(* LS Electric XG5000 project: XEM_iX7_ModTCP_Example *)
(* PLC LSPLC *)
(* module base 0 slot 0: Input/Output Module:XEM-DN/DP32HP (DC 24V Input, Transistor Output, 32 Contacts) *)
(* module base 0 slot 1: Internal Positioning:XBF-PO06E (Open Collector Type, 6 Axis) *)
VAR_GLOBAL
    gControl_Word AT %MW1 : WORD; (* global control word for controlling the iX7 over Modbus TCP *)
    gStatus_Word AT %MW2 : WORD; (* global status word data for iX7 drive over Modbus TCP *)
    gSV_ON AT %MX0 : BOOL; (* global Command to turn servo on/off sent over Modbus RTU *)
    gTarget_Position AT %MW3 : ARRAY[0..1] OF WORD; (* global target position in an array of words *)
    gVelocity_Accel_Decel AT %MW4 : ARRAY[0..5] OF WORD; (* word array for setting up velocity, acceleration and deceleration of the modbus TCP move *)
END_VAR

PROGRAM NewProgram (* task: Scan Program *)
VAR
    Acceleration : DINT; (* acceleration of the move *)
    Deceleration : DINT; (* deceleration of the move *)
    Halt_Motion : BOOL; (* halt motion of the modbus servo *)
    Move_Type0 : BOOL; (* Move type 0 is wait until current move is complete *)
    Move_Type1 : BOOL; (* move to target position immediately *)
    Move_Type2 : BOOL; (* Drives from the current position to the profile position at the profile / velocity before it applies the next position. *)
    Positioning_Mode : BOOL; (* False = Absolute Positioning; True = Relative Positioning *)
    Servo_Enable : BOOL; (* Enable servo - local command to enable servos *)
    Start_Motion : BOOL; (* local command to start motion *)
    Target_Position : DINT; (* local index01 distance value *)
    tempDword : DWORD; (* temporary dword storage *)
    Velocity : DINT; (* velocity of the move *)
END_VAR
VAR_EXTERNAL
    gControl_Word : WORD; (* AT %MW1 *) (* global control word for controlling the iX7 over Modbus TCP *)
    gStatus_Word : WORD; (* AT %MW2 *) (* global status word data for iX7 drive over Modbus TCP *)
    gSV_ON : BOOL; (* AT %MX0 *) (* global Command to turn servo on/off sent over Modbus RTU *)
    gTarget_Position : ARRAY[0..1] OF WORD; (* AT %MW3 *) (* global target position in an array of words *)
    gVelocity_Accel_Decel : ARRAY[0..5] OF WORD; (* AT %MW4 *) (* word array for setting up velocity, acceleration and deceleration of the modbus TCP move *)
END_VAR

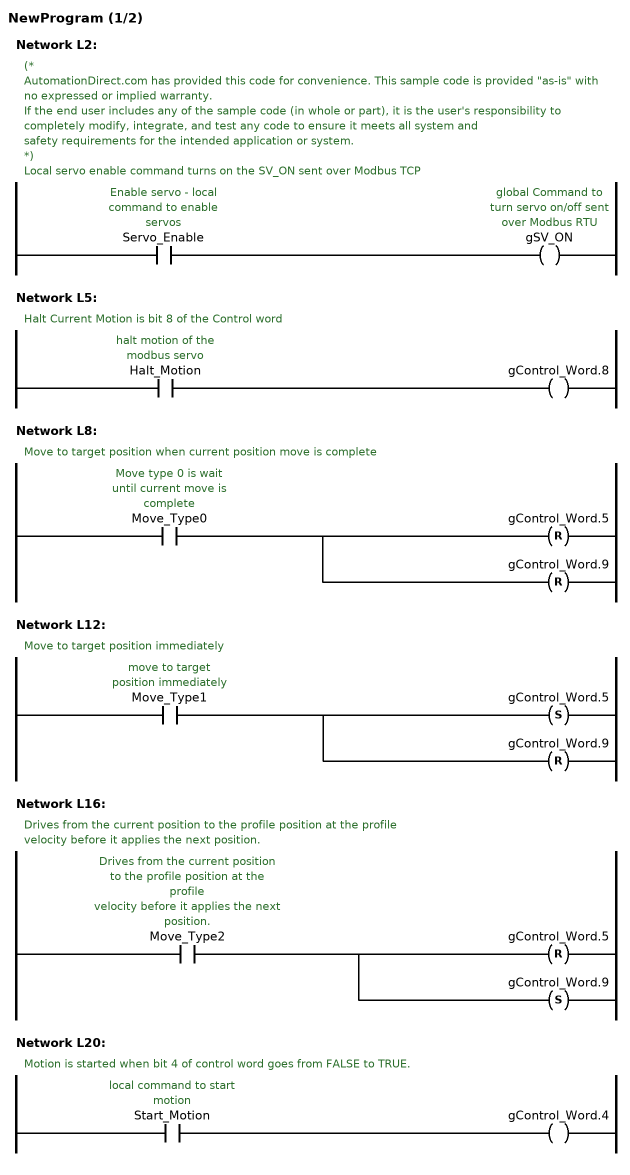
(* ( * / AutomationDirect.com has provided this code for convenience. This sample code is provided "as-is" with no expressed or implied warranty. / If the end user includes any of the sample code (in whole or part), it is the user's responsibility to completely modify, integrate, and test any code to ensure it meets all system and / safety requirements for the intended application or system. / * ) *)
(* Local servo enable command turns on the SV_ON sent over Modbus TCP *)
(* Rung L2 *)
gSV_ON := Servo_Enable;
(* Halt Current Motion is bit 8 of the Control word *)
(* Rung L5 *)
gControl_Word.8 := Halt_Motion;
(* Move to target position when current position move is complete *)
(* Rung L8 *)
IF Move_Type0 THEN
    gControl_Word.5 := FALSE;
    gControl_Word.9 := FALSE;
END_IF;
(* Move to target position immediately *)
(* Rung L12 *)
IF Move_Type1 THEN
    gControl_Word.5 := TRUE;
    gControl_Word.9 := FALSE;
END_IF;
(* Drives from the current position to the profile position at the profile / velocity before it applies the next position. *)
(* Rung L16 *)
IF Move_Type2 THEN
    gControl_Word.5 := FALSE;
    gControl_Word.9 := TRUE;
END_IF;
(* Motion is started when bit 4 of control word goes from FALSE to TRUE. *)
(* Rung L20 *)
gControl_Word.4 := Start_Motion;

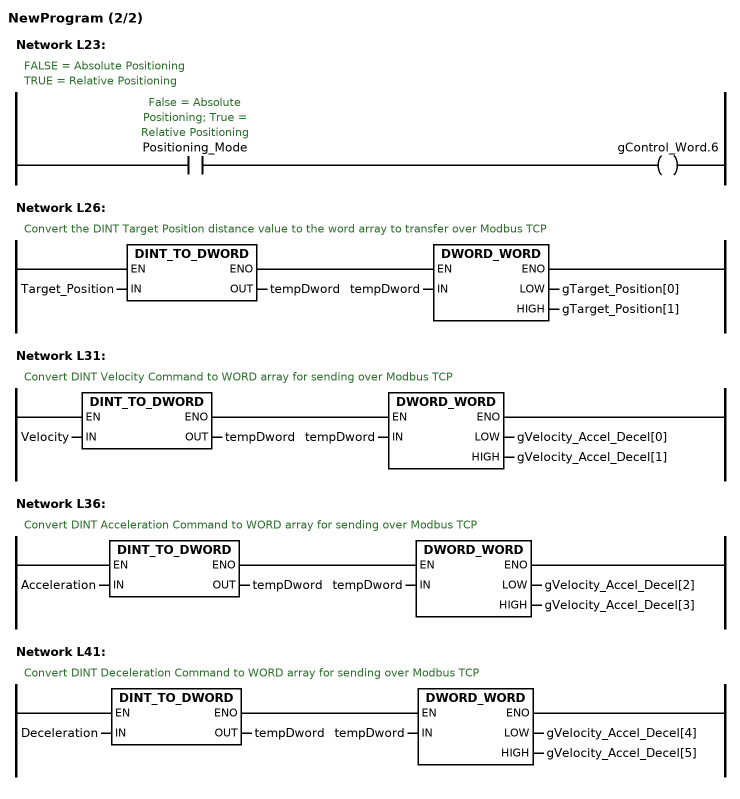
(* FALSE = Absolute Positioning / TRUE = Relative Positioning *)
(* Rung L23 *)
gControl_Word.6 := Positioning_Mode;
(* Convert the DINT Target Position distance value to the word array to transfer over Modbus TCP *)
(* Rung L26 *)
tempDword := DINT_TO_DWORD(Target_Position);
gTarget_Position[0] := DWORD_WORD(IN := tempDword, HIGH => gTarget_Position[1]);
(* Convert DINT Velocity Command to WORD array for sending over Modbus TCP *)
(* Rung L31 *)
tempDword := DINT_TO_DWORD(Velocity);
gVelocity_Accel_Decel[0] := DWORD_WORD(IN := tempDword, HIGH => gVelocity_Accel_Decel[1]);
(* Convert DINT Acceleration Command to WORD array for sending over Modbus TCP *)
(* Rung L36 *)
tempDword := DINT_TO_DWORD(Acceleration);
gVelocity_Accel_Decel[2] := DWORD_WORD(IN := tempDword, HIGH => gVelocity_Accel_Decel[3]);
(* Convert DINT Deceleration Command to WORD array for sending over Modbus TCP *)
(* Rung L41 *)
tempDword := DINT_TO_DWORD(Deceleration);
gVelocity_Accel_Decel[4] := DWORD_WORD(IN := tempDword, HIGH => gVelocity_Accel_Decel[5]);
END_PROGRAM